// TIA Portal V20 export
DATA_BLOCK "ErrCom_DB"   // DB303
// stored: AutoNumber false, InstanceOfName ErrCom, InstanceOfType FB
"ErrCom"
   // VAR
   //    Var { S7_SetPoint := 'True'} : "TypeVar";
   //    T : Array[1..1] of IEC_TIMER;
   // END_VAR
BEGIN
END_DATA_BLOCK
